// §14 under test: F_Sha256 against the FIPS 180-4 example vectors - the empty
// message, one block, and a message whose padding spills into a second block.
FUNCTION_BLOCK FB_Sha256_Tests EXTENDS TcUnit.FB_TestSuite
VAR
    _digest : ARRAY[0..31] OF BYTE;
END_VAR

The_empty_message_hashes_to_the_published_digest();
One_block_hashes_to_the_published_digest();
Two_blocks_hash_to_the_published_digest();

// The digest of Text as 64 lowercase hex characters.
METHOD PRIVATE _M_Hex : STRING(64)
VAR_INPUT
    Text : STRING(80);
END_VAR
VAR
    i : INT;
    nib : BYTE;
    hex : STRING(16) := '0123456789abcdef';
    out : STRING(64);
    pOut : POINTER TO BYTE;
    pHex : POINTER TO BYTE;
END_VAR
F_Sha256(pData := ADR(Text), Size := INT_TO_UDINT(LEN(Text)), Digest := _digest);
pOut := ADR(out);
pHex := ADR(hex);
FOR i := 0 TO 31 DO
    nib := SHR(_digest[i], 4);
    pOut[2 * i] := pHex[nib];
    nib := _digest[i] AND 16#0F;
    pOut[2 * i + 1] := pHex[nib];
END_FOR
pOut[64] := 0;
_M_Hex := out;
END_METHOD

METHOD The_empty_message_hashes_to_the_published_digest
TEST('The_empty_message_hashes_to_the_published_digest');
AssertEquals_STRING(
    Expected := 'e3b0c44298fc1c149afbf4c8996fb92427ae41e4649b934ca495991b7852b855',
    Actual := _M_Hex(Text := ''), Message := 'SHA-256 of the empty message');
TEST_FINISHED();
END_METHOD

METHOD One_block_hashes_to_the_published_digest
TEST('One_block_hashes_to_the_published_digest');
AssertEquals_STRING(
    Expected := 'ba7816bf8f01cfea414140de5dae2223b00361a396177a9cb410ff61f20015ad',
    Actual := _M_Hex(Text := 'abc'), Message := 'SHA-256 of abc');
TEST_FINISHED();
END_METHOD

METHOD Two_blocks_hash_to_the_published_digest
TEST('Two_blocks_hash_to_the_published_digest');
AssertEquals_STRING(
    Expected := '248d6a61d20638b8e5c026930c3e6039a33ce45964ff2167f6ecedd419db06c1',
    Actual := _M_Hex(Text := 'abcdbcdecdefdefgefghfghighijhijkijkljklmklmnlmnomnopnopq'),
    Message := 'SHA-256 of the 56-byte FIPS message (padding needs a second block)');
TEST_FINISHED();
END_METHOD

END_FUNCTION_BLOCK

(* stored: Version 1.1.0.1, ProductVersion 3.1.4024.12
   POU FB_Sha256_Tests: Id {fc2bc675-8364-444d-ae3d-e13b6b4d288f}, SpecialFunc None
   Method _M_Hex: Id {0da5dfb8-69d1-4173-9377-52d3e479765a}
   Method The_empty_message_hashes_to_the_published_digest: Id {ee661187-0185-48c5-bf66-e5d34788a927}
   Method One_block_hashes_to_the_published_digest: Id {622ab1a2-1503-4b1d-993e-def718ba7c44}
   Method Two_blocks_hash_to_the_published_digest: Id {f15cd7b9-f3b0-41ca-89e4-1a9212410cf0} *)
